TYPE ST_LaudaReadCommands_ControlParameters :
STRUCT
END_STRUCT
END_TYPE

(* stored: Version 1.1.0.1, ProductVersion 3.1.4024.13
   DUT ST_LaudaReadCommands_ControlParameters: Id {756b1bdb-0fa0-437e-874a-fefa4f10b5f5} *)
